{attribute 'pack_mode' := '1'}
TYPE ST_MsgToCCS EXTENDS ST_PLCMsg:
STRUCT
	sequence: DINT;(* Increment this to ensure notification. *)
END_STRUCT
END_TYPE

(* stored: Version 1.1.0.1, ProductVersion 3.1.4020.12
   DUT ST_MsgToCCS: Id {d9adaf84-3e96-4a0a-8a6d-4dff4db760ca} *)
